{attribute addProperty BoxType "BK1250-0000-0000"}
{attribute addProperty Id "InputsAT %I*Inputs_6F058048000OutputsAT %I*Outputs_9C14F798000WcStateAT %I*WcState_98A4DF7520.250InfoDataAT %I*InfoData_275E3363128160"}
{attribute addProperty CRC "1783375152"}
{attribute addProperty SizeInBites "130"}
{attribute addProperty SizeInBytes "16.25"}
TYPE BK1250_4487A81F :
STRUCT
	{attribute addProperty Name "Inputs"}
	Inputs : Inputs_6F058048;
	{attribute addProperty Name "Outputs"}
	Outputs : Outputs_9C14F798;
	{attribute addProperty Name "WcState"}
	WcState : WcState_98A4DF75;
	{attribute addProperty Name "InfoData"}
	InfoData : InfoData_275E3363;
END_STRUCT
END_TYPE

(* stored: Version 1.2.0.0, ProductVersion 3.1.4024.9
   DUT BK1250_4487A81F: Id {56668a80-ade2-4116-8f46-191828e5d6b8} *)
